// Mitsubishi GX Works2 project: PID_TEST_SIMKORT_V7   PLC: FX2N/FX2NC

// global labels: Global1
VAR_GLOBAL
  Process_val AT D0 : REAL;
  Reference AT D2 : REAL;
  U_Nominal_Intouch AT D4 : REAL;
  Controller_Out AT D6 : REAL;
  P_Mode_Intouch AT D8 : REAL;
  PI_Mode_Intouch AT D10 : REAL;
  PD_Mode_Intouch AT D12 : REAL;
  PID_Mode_Intouch AT D14 : REAL;
  Manual_Mode_Intouch AT D16 : REAL;
  Kp_Intouch AT D18 : REAL;
  Ti_Intouch AT D20 : REAL;
  Td_Intouch AT D22 : REAL;
END_VAR
VAR_GLOBAL CONSTANT
  Sampling_Interval : REAL := 0.1;
  Filter_Constant_Intouch : REAL := 10.0;
END_VAR
VAR_GLOBAL
  FeedForward_OnOff_Intouch AT D26 : REAL;
  FeedForward_Output AT D44 : REAL;
  Kff_Intouch AT D28 : REAL;
  Tau_Lead_Intouch AT D30 : REAL;
  Tau_Lag_Intouch AT D32 : REAL;
  Disturbance_Intouch AT D34 : REAL;
  Filtered_Disturbance AT D40 : REAL;
  Antiwindup_OnOff_Intouch AT D42 : REAL;
  Feed_Forward AT D36 : REAL;
  Utot AT D38 : REAL;
END_VAR
VAR_GLOBAL CONSTANT
  Umax_PID : REAL := 100.0;
  Umin_PID : REAL;
  Max_ChangeRate_PID : REAL := 100.0;
  Min_ChangeRate_PID : REAL := -100.0;
  Tracking_coeff : REAL := 1.5;
  Kb_Intouch : REAL := 2;
  Kt_Intouch : REAL := 2;
END_VAR
VAR_GLOBAL
  PID_Proportional_Output AT D46 : REAL;
  PID_Integral_Output AT D48 : REAL;
  PID_Derivative_Output AT D50 : REAL;
END_VAR

// task Task_01 (event FALSE, interval T#100ms, priority 31): POU_01

PROGRAM POU_01
VAR
  PID_Controller_1 : PID_Controller;
  TestProsess_1 : TestProsess;
  Linear_Interpolation_1 : Linear_Interpolation;
  Linear_Interpolation_2 : Linear_Interpolation;
  LP_Filter_1 : LP_Filter;
  LeadLag_1 : LeadLag;
  Rate_Limiter_1 : Rate_Limiter;
  Controller_Options_1 : Controller_Options;
  Linear_Interpolation_3 : Linear_Interpolation;
  Linear_Interpolation_4 : Linear_Interpolation;
  Saturation_1 : Saturation;
  PID_Output_Options_1 : PID_Output_Options;
  Integrator_Init : REAL;
  PID_Output : REAL;
END_VAR
(* structured ladder/FBD written out as ST: instructions are called as NAME(EN, inputs, outputs); _pN, _eN, _tN stand for wires *)
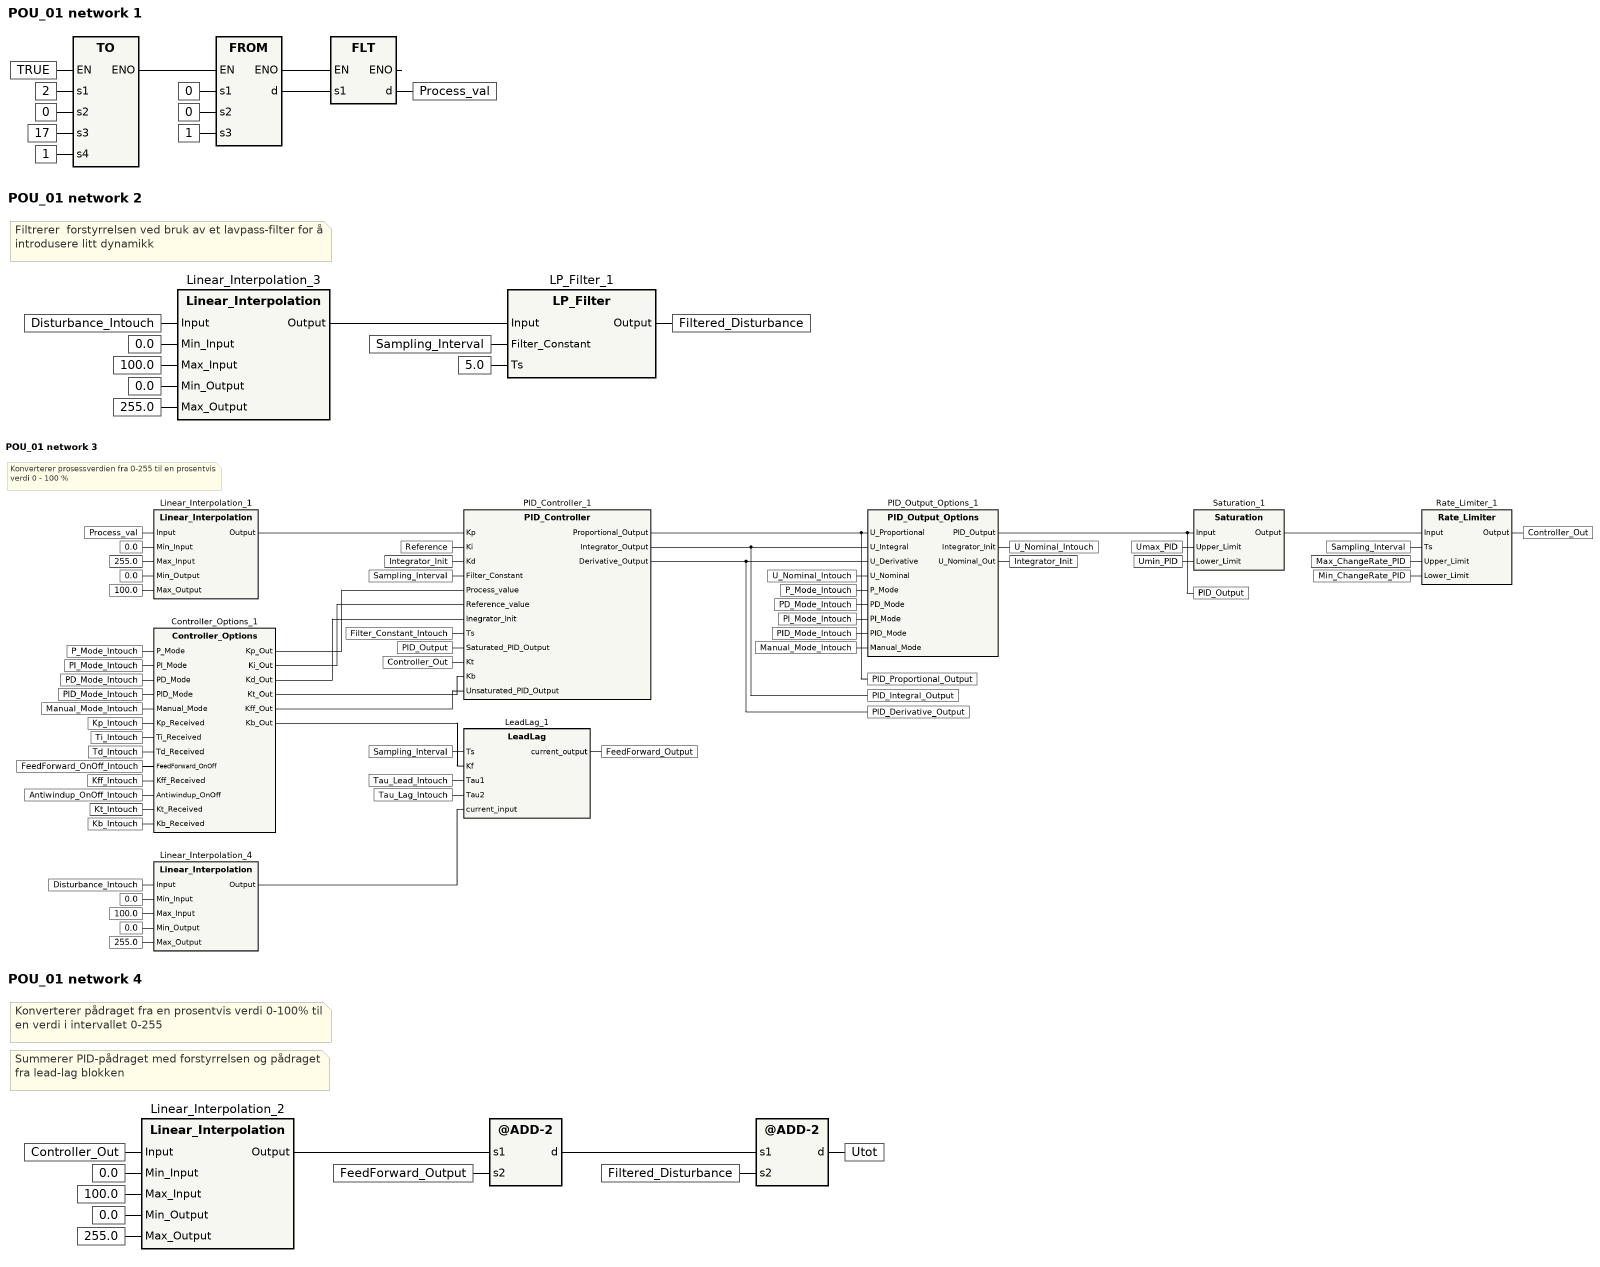
(* network 1 *)
_e1 := TO(TRUE, 2, 0, 17, 1);
_e3 := FROM(_e1, 0, 0, 1, _t2);
FLT(_e3, _t2, Process_val);
(* network 2 *)
(* Filtrerer  forstyrrelsen ved bruk av et lavpass-filter for å introdusere litt dynamikk *)
Linear_Interpolation_3(Input := Disturbance_Intouch, Min_Input := 0.0, Max_Input := 100.0, Min_Output := 0.0, Max_Output := 255.0);
LP_Filter_1(Input := Linear_Interpolation_3.Output, Filter_Constant := Sampling_Interval, Ts := 5.0, Output => Filtered_Disturbance);
(* network 3 *)
(* Konverterer prosessverdien fra 0-255 til en prosentvis verdi 0 - 100 % *)
Linear_Interpolation_1(Input := Process_val, Min_Input := 0.0, Max_Input := 255.0, Min_Output := 0.0, Max_Output := 100.0);
Controller_Options_1(P_Mode := P_Mode_Intouch, PI_Mode := PI_Mode_Intouch, PD_Mode := PD_Mode_Intouch, PID_Mode := PID_Mode_Intouch, Manual_Mode := Manual_Mode_Intouch, Kp_Received := Kp_Intouch, Ti_Received := Ti_Intouch, Td_Received := Td_Intouch, FeedForward_OnOff := FeedForward_OnOff_Intouch, Kff_Received := Kff_Intouch, Antiwindup_OnOff := Antiwindup_OnOff_Intouch, Kt_Received := Kt_Intouch, Kb_Received := Kb_Intouch);
PID_Controller_1(Kp := Linear_Interpolation_1.Output, Ki := Reference, Kd := Integrator_Init, Filter_Constant := Sampling_Interval, Process_value := Controller_Options_1.Kp_Out, Reference_value := Controller_Options_1.Ki_Out, Inegrator_Init := Controller_Options_1.Kd_Out, Ts := Filter_Constant_Intouch, Saturated_PID_Output := PID_Output, Kt := Controller_Out, Kb := Controller_Options_1.Kt_Out, Unsaturated_PID_Output := Controller_Options_1.Kff_Out);
PID_Proportional_Output := PID_Controller_1.Proportional_Output;
PID_Integral_Output := PID_Controller_1.Integrator_Output;
PID_Derivative_Output := PID_Controller_1.Derivative_Output;
PID_Output_Options_1(U_Proportional := PID_Controller_1.Proportional_Output, U_Integral := PID_Controller_1.Integrator_Output, U_Derivative := PID_Controller_1.Derivative_Output, U_Nominal := U_Nominal_Intouch, P_Mode := P_Mode_Intouch, PD_Mode := PD_Mode_Intouch, PI_Mode := PI_Mode_Intouch, PID_Mode := PID_Mode_Intouch, Manual_Mode := Manual_Mode_Intouch, Integrator_Init => U_Nominal_Intouch, U_Nominal_Out => Integrator_Init);
PID_Output := PID_Output_Options_1.PID_Output;
Saturation_1(Input := PID_Output_Options_1.PID_Output, Upper_Limit := Umax_PID, Lower_Limit := Umin_PID);
Rate_Limiter_1(Input := Saturation_1.Output, Ts := Sampling_Interval, Upper_Limit := Max_ChangeRate_PID, Lower_Limit := Min_ChangeRate_PID, Output => Controller_Out);
Linear_Interpolation_4(Input := Disturbance_Intouch, Min_Input := 0.0, Max_Input := 100.0, Min_Output := 0.0, Max_Output := 255.0);
LeadLag_1(Ts := Sampling_Interval, Kf := Controller_Options_1.Kb_Out, Tau1 := Tau_Lead_Intouch, Tau2 := Tau_Lag_Intouch, current_input := Linear_Interpolation_4.Output, current_output => FeedForward_Output);
(* network 4 *)
(* Konverterer pådraget fra en prosentvis verdi 0-100% til en verdi i intervallet 0-255 *)
(* Summerer PID-pådraget med forstyrrelsen og pådraget fra lead-lag blokken *)
Linear_Interpolation_2(Input := Controller_Out, Min_Input := 0.0, Max_Input := 100.0, Min_Output := 0.0, Max_Output := 255.0);
Utot := @ADD-2(@ADD-2(Linear_Interpolation_2.Output, FeedForward_Output), Filtered_Disturbance);
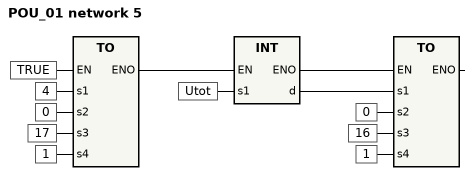
(* network 5 *)
_e1 := TO(TRUE, 4, 0, 17, 1);
_e3 := INT(_e1, Utot, _t2);
TO(_e3, _t2, 0, 16, 1);
END_PROGRAM

FUNCTION_BLOCK PID_Controller
VAR_INPUT
  Kp : REAL;  (* Proportional gain *)
  Ki : REAL;  (* Integral coefficient ( I = 1/Ti ) *)
  Kd : REAL;  (* Derivative coefficient ( D = Td ) *)
  Filter_Constant : REAL;  (* Filter constant N *)
  Process_value : REAL;
  Reference_value : REAL;
  Inegrator_Init : REAL;
  Ts : REAL;  (* Sampling time *)
END_VAR
VAR
  Integrator_OnOff : REAL;  (* Turn integrator On (1) or Off (0) *)
END_VAR
VAR_INPUT
  Saturated_PID_Output : REAL;
  Kt : REAL;
  Kb : REAL;
END_VAR
VAR
  MUL3_1 : MUL3;
  ADD4_1 : ADD4;
  Derivate_BackDiff_1 : Derivate_BackDiff;
  Integrate_Tustin_1 : Integrate_Tustin;
  LP_Filter_1 : LP_Filter;
  Integrator_Options_1 : Integrator_Options;
  Rate_Limiter_1 : Rate_Limiter;
END_VAR
VAR_OUTPUT
  Proportional_Output : REAL;
END_VAR
VAR_INPUT
  Unsaturated_PID_Output : REAL;
END_VAR
VAR_OUTPUT
  Integrator_Output : REAL;
  Derivative_Output : REAL;
END_VAR
(* structured ladder/FBD written out as ST: instructions are called as NAME(EN, inputs, outputs); _pN, _eN, _tN stand for wires *)
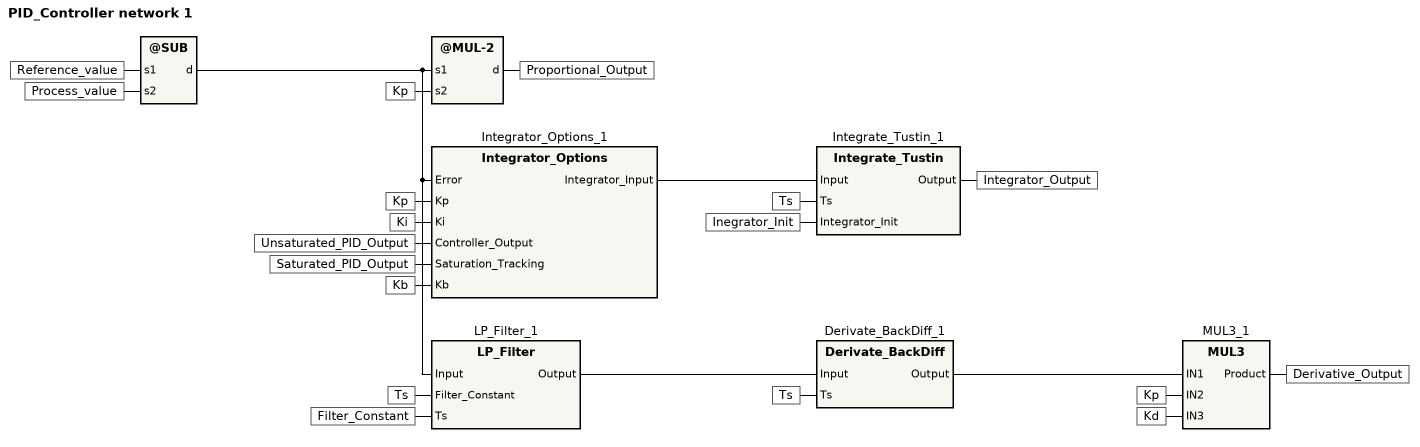
(* network 1 *)
_p1 := @SUB(Reference_value, Process_value);
Proportional_Output := @MUL-2(_p1, Kp);
Integrator_Options_1(Error := _p1, Kp := Kp, Ki := Ki, Controller_Output := Unsaturated_PID_Output, Saturation_Tracking := Saturated_PID_Output, Kb := Kb);
Integrate_Tustin_1(Input := Integrator_Options_1.Integrator_Input, Ts := Ts, Integrator_Init := Inegrator_Init, Output => Integrator_Output);
LP_Filter_1(Input := _p1, Filter_Constant := Ts, Ts := Filter_Constant);
Derivate_BackDiff_1(Input := LP_Filter_1.Output, Ts := Ts);
MUL3_1(IN1 := Derivate_BackDiff_1.Output, IN2 := Kp, IN3 := Kd, Product => Derivative_Output);
END_FUNCTION_BLOCK

FUNCTION_BLOCK LP_Filter
VAR_INPUT
  Input : REAL;
END_VAR
VAR_OUTPUT
  Output : REAL;
END_VAR
VAR
  Previous_Output : REAL;
END_VAR
VAR_INPUT
  Filter_Constant : REAL;
END_VAR
VAR
  Beta : REAL;
END_VAR
VAR_INPUT
  Ts : REAL;
END_VAR
Beta := Filter_Constant*Ts / ( 1.0 + Filter_Constant*Ts) ;

Output := Beta*Input + (1.0 - Beta) * Previous_Output;

Previous_Output := Output;
END_FUNCTION_BLOCK

FUNCTION_BLOCK Derivate_BackDiff
VAR_INPUT
  Input : REAL;
END_VAR
VAR
  Previous_Input : REAL;
END_VAR
VAR_OUTPUT
  Output : REAL;
END_VAR
VAR_INPUT
  Ts : REAL;
END_VAR
Output := (Input - Previous_Input) / Ts;

Previous_Input := Input;
END_FUNCTION_BLOCK

FUNCTION_BLOCK MUL3
VAR_INPUT
  IN1 : REAL;
  IN2 : REAL;
  IN3 : REAL;
END_VAR
VAR_OUTPUT
  Product : REAL;
END_VAR
Product := IN1 * IN2 * IN3;
END_FUNCTION_BLOCK

FUNCTION_BLOCK ADD4
VAR_INPUT
  IN1 : REAL;
  IN2 : REAL;
  IN3 : REAL;
  IN4 : REAL;
END_VAR
VAR_OUTPUT
  SUM4 : REAL;
END_VAR
VAR_INPUT
  Kp : REAL;
END_VAR
VAR_OUTPUT
  Proposjonal : REAL;
  Integral : REAL;
  Derivat : REAL;
END_VAR
VAR_INPUT
  Ki : REAL;
END_VAR

Proposjonal := IN2;
Integral := IN3;
Derivat := IN4;

IF (Ki = 0.0) THEN; 
	Integral := 0.0;
END_IF;

IF (Kp = 0.0) THEN;
	SUM4 := IN1;
	
ELSE;
	SUM4 := IN1 + Proposjonal+ Integral+ Derivat;
END_IF;
END_FUNCTION_BLOCK

FUNCTION_BLOCK TestProsess
VAR_INPUT
  Ts : REAL;  (* Sampling period *)
  Gain : REAL;  (* Process gain *)
  Tau : REAL;  (* Process time-constant *)
  Zeta : REAL;  (* Damping ratio (?) *)
END_VAR
VAR
  Outputs : ARRAY [0..2] OF REAL;  (* Array containing current -and previous output *)
  Inputs : ARRAY [0..2] OF REAL;  (* Array containing current -and previous input *)
END_VAR
VAR_INPUT
  current_input : REAL;
END_VAR
VAR_OUTPUT
  current_output : REAL;
END_VAR
Inputs[2] := current_input;

Outputs[2] := ( Outputs[1]*(8.0*Tau*Tau-2.0*Ts*Ts) + Outputs[0]*(4.0*Zeta*Tau*Ts-4.0*Tau*Tau-Ts*Ts) + Inputs[2]*Gain*Ts*Ts + Inputs[1]*2.0*Gain*Ts*Ts+Inputs[0]*Gain*Ts*Ts )  /  ( 4.0*Tau*Tau+4.0*Zeta*Tau*Ts+Ts*Ts );
current_output := Outputs[2];

Inputs[0] := Inputs[1];
Inputs[1] := Inputs[2];

Outputs[0] := Outputs[1];
Outputs[1] := Outputs[2];
END_FUNCTION_BLOCK

FUNCTION_BLOCK Integrate_Tustin
VAR_INPUT
  Input : REAL;
END_VAR
VAR
  Previous_Input : REAL;
END_VAR
VAR_OUTPUT
  Output : REAL;
END_VAR
VAR
  Previous_Output : REAL;
END_VAR
VAR_INPUT
  Ts : REAL;
  Integrator_Init : REAL;
END_VAR
VAR
  Prev_Integrator_Init : REAL;
END_VAR
IF ( Integrator_Init <> Prev_Integrator_Init) THEN; (* Reset integrator to initializer value *)
	Output := Integrator_Init;
ELSE;
	Output := ( Previous_Output + Ts*( Input + Previous_Input ) / (2.0) );
END_IF;

Prev_Integrator_Init := Integrator_Init;

Previous_Input := Input;
Previous_Output := Output;
END_FUNCTION_BLOCK

FUNCTION_BLOCK Integrator_Options
VAR_INPUT
  Error : REAL;  (* Reference - ProcessValue *)
  Kp : REAL;  (* Proportional Gain *)
  Ki : REAL;  (* Integral Gain *)
END_VAR
VAR_OUTPUT
  Integrator_Input : REAL;
END_VAR
VAR_INPUT
  Controller_Output : REAL;  (* Output of PID-controller *)
  Saturation_Tracking : REAL;
  Kb : REAL;
END_VAR
Integrator_Input := Error*Kp*Ki + (Saturation_Tracking - Controller_Output) * Kb ;
END_FUNCTION_BLOCK

FUNCTION_BLOCK Saturation
VAR_INPUT
  Input : REAL;
  Upper_Limit : REAL;
  Lower_Limit : REAL;
END_VAR
VAR_OUTPUT
  Output : REAL;
END_VAR
Output := Input;

IF ( Input > Upper_Limit ) THEN
	Output := Upper_Limit;
END_IF;

IF Input < Lower_Limit THEN
	Output := Lower_Limit;
END_IF;
END_FUNCTION_BLOCK

FUNCTION_BLOCK Rate_Limiter
VAR_INPUT
  Input : REAL;
  Ts : REAL;
  Upper_Limit : REAL;
  Lower_Limit : REAL;
END_VAR
VAR_OUTPUT
  Output : REAL;
END_VAR
VAR
  Rate : REAL;
  Previous_Output : REAL;
END_VAR
Rate := ( Input - Previous_Output ) / Ts;

Output := Input;

IF ( Rate > Upper_Limit) THEN
	Output := Previous_Output + Upper_Limit*Ts;
END_IF;

IF ( Rate < Lower_Limit) THEN
	Output := Previous_Output + Lower_Limit*Ts;
END_IF;

Previous_Output := Output;
END_FUNCTION_BLOCK

FUNCTION_BLOCK Linear_Interpolation
VAR_INPUT
  Input : REAL;
  Min_Input : REAL;
  Max_Input : REAL;
  Min_Output : REAL;
  Max_Output : REAL;
END_VAR
VAR_OUTPUT
  Output : REAL;
END_VAR
Output := Min_Output + (Input - Min_Input) * (Max_Output - Min_Output) / (Max_Input - Min_Input );
END_FUNCTION_BLOCK

FUNCTION_BLOCK LeadLag
VAR_INPUT
  Ts : REAL;  (* Sampling period *)
  Kf : REAL;  (* Lead-Lag Unit gain *)
  Tau1 : REAL;  (* Numerator time-constant *)
  Tau2 : REAL;  (* Denominator time-constant *)
END_VAR
VAR
  Outputs : ARRAY [0..1] OF REAL;  (* Array containing current -and previous output *)
  Inputs : ARRAY [0..1] OF REAL;  (* Array containing current -and previous input *)
END_VAR
VAR_INPUT
  current_input : REAL;
END_VAR
VAR_OUTPUT
  current_output : REAL;
END_VAR
Inputs[1] := current_input;

Outputs[1] := ( ( 2.0*Tau2-Ts)*Outputs[0] + Kf*(2.0*Tau1+Ts)*Inputs[1] + Kf*(Ts-2.0*Tau1)*Inputs[0] ) / (2.0*Tau2+Ts);
current_output := Outputs[1];

Inputs[0] := Inputs[1];
Outputs[0] := Outputs[1];
END_FUNCTION_BLOCK

FUNCTION_BLOCK Controller_Options
VAR_INPUT
  P_Mode : REAL;
  PI_Mode : REAL;
  PD_Mode : REAL;
  PID_Mode : REAL;
  Manual_Mode : REAL;
  Kp_Received : REAL;
  Ti_Received : REAL;
  Td_Received : REAL;
  FeedForward_OnOff : REAL;
  Kff_Received : REAL;
END_VAR
VAR_OUTPUT
  Kp_Out : REAL;
  Ki_Out : REAL;
  Kd_Out : REAL;
  Kt_Out : REAL;
END_VAR
VAR_INPUT
  Antiwindup_OnOff : REAL;
  Kt_Received : REAL;
END_VAR
VAR_OUTPUT
  Kff_Out : REAL;
END_VAR
VAR_INPUT
  Kb_Received : REAL;
END_VAR
VAR_OUTPUT
  Kb_Out : REAL;
END_VAR
IF ( P_Mode = 1.0 ) THEN;
	Kp_Out := Kp_Received;
	Ki_Out := 0.0;
	Kd_Out := 0.0;

ELSIF ( PI_Mode = 1.0 ) THEN;
	Kp_Out := Kp_Received;
	Ki_Out := 1.0/Ti_Received;
	Kd_Out := 0.0;

ELSIF ( PD_Mode = 1.0 ) THEN;
	Kp_Out := Kp_Received;
	Ki_Out := 0.0;
	Kd_Out :=Td_Received;

ELSIF ( PID_Mode = 1.0 ) THEN;
	Kp_Out := Kp_Received;
	Ki_Out := 1.0/Ti_Received;
	Kd_Out :=Td_Received;

ELSIF ( Manual_Mode = 1.0 ) THEN;
	Kp_Out := 0.0;
	Ki_Out := 0.0;
	Kd_Out :=0.0;

END_IF;

IF ( FeedForward_OnOff = 1.0 ) THEN;
	Kff_Out := Kff_Received;
ELSE;
	Kff_Out := 0.0;
END_IF;

IF (Ki_Out> 0.0 ) THEN;
	Kt_Out:= 0.0;
ELSE;
	Kt_Out := Kt_Received;
END_IF;

IF ( Antiwindup_OnOff = 1.0 ) THEN;
	Kb_Out := Kb_Received;
ELSE;
	Kb_Out := 0.0;
END_IF;
END_FUNCTION_BLOCK

FUNCTION_BLOCK PID_Output_Options
VAR_INPUT
  U_Proportional : REAL;
  U_Integral : REAL;
  U_Derivative : REAL;
  U_Nominal : REAL;
  P_Mode : REAL;
  PD_Mode : REAL;
  PI_Mode : REAL;
  PID_Mode : REAL;
  Manual_Mode : REAL;
END_VAR
VAR
  Prev_P_Mode : REAL;
  Prev_PD_Mode : REAL;
  Prev_PI_Mode : REAL;
  Prev_PID_Mode : REAL;
  Prev_Manual_Mode : REAL;
  Prev_U_Nominal : REAL;
END_VAR
VAR_OUTPUT
  PID_Output : REAL;
  Integrator_Init : REAL;
  U_Nominal_Out : REAL;
END_VAR
VAR
  Prev_PID_Output : REAL;
  Count : REAL;
END_VAR


IF (Prev_Manual_Mode = 1.0 AND (PI_Mode = 1.0 OR PID_Mode = 1.0) ) THEN; (* Switch from manual to controller with integrator *)
	Integrator_Init := Prev_PID_Output - U_Proportional;
	
ELSIF ( (Prev_P_Mode = 1.0 OR Prev_PD_Mode = 1.0) AND  (PI_Mode = 1.0 OR PID_Mode = 1.0) ) THEN;
	Integrator_Init := Prev_U_Nominal;
	
ELSIF ( P_Mode = 1.0) THEN;
	PID_Output := U_Nominal + U_Proportional;

ELSIF ( PI_Mode = 1.0 ) THEN;
	PID_Output := U_Proportional + U_Integral;

ELSIF ( PD_Mode = 1.0 ) THEN;
	PID_Output := U_Nominal + U_Proportional + U_Derivative;

ELSIF ( PID_Mode = 1.0 ) THEN;
	PID_Output := U_Proportional + U_Integral + U_Derivative;

ELSIF ( Manual_Mode = 1.0 ) THEN;
	PID_Output := U_Nominal;
END_IF;

Prev_U_Nominal := U_Nominal;

Prev_PID_Output := PID_Output;
Prev_Manual_Mode := Manual_Mode;
Prev_PD_Mode := PD_Mode;
Prev_PI_Mode := PI_Mode;
Prev_PID_Mode := PID_Mode;
Prev_P_Mode := P_Mode;
END_FUNCTION_BLOCK
